(* PLC project PLC_Rack, Beckhoff Automation GmbH TwinCAT PLC Control 3.5.13.21 *)
(* stored: creationDateTime 2025-07-11T10:35:19.1083173, modificationDateTime 2025-07-11T10:35:19.1104652 *)

PROGRAM MAIN
VAR
	// Input Variable
	bS10 AT%I*: BOOL;				// Schalter S10
	bS11 AT%I*: BOOL;				// Schalter S11
	bS12 AT%I*: BOOL;				// Schalter S12
	
	// Output Variable
	bL10 		AT%Q*	: BOOL;		// LED S10
	bL11 		AT%Q*	: BOOL;		// LED S11
	bL12 		AT%Q*	: BOOL;		// LED S12
	bL13 		AT%Q*	: BOOL;		// LED S13
	nCount		AT%Q*	: LREAL;	// Zählvariable
	
	// Timer
	ton1	: TON;
	ton2	: TON;
	ton3	: TON;
	
	// Zähler
	ctud	: CTUD;
	
	// Trigger
	rTrig	: R_TRIG;
	fTrig	: F_TRIG;
	
END_VAR

            // Hier den Code ändern

// TASTER
	// Counter erhöhen, wenn Taster S10 gedrückt
	IF bS10 THEN
		nCount := LIMIT(0,nCount + 1,10);
	END_IF
	// Counter verringern, wenn Taster S11 gedrückt
	IF bS11 THEN
		nCount := LIMIT(0,nCount - 1,10);
	END_IF

// LEDs
	bL10 := bS10;
	bL11 := bS10;
	bL12 := bS10;
	bL13 := bS10;
	
	
	


          
END_PROGRAM
